INTERFACE ITF_Filling EXTENDS ITF_PackML

{warning 'add method implementation '}
METHOD Abort : BOOL
END_METHOD

{warning 'add method implementation '}
METHOD Aborting_SC : BOOL
END_METHOD

{warning 'add method implementation '}
METHOD Clear : BOOL
END_METHOD

{warning 'add method implementation '}
METHOD Clearing_SC : BOOL
END_METHOD

{warning 'add method implementation '}
METHOD Completing_SC : BOOL
END_METHOD

{warning 'add method implementation '}
METHOD Execute_SC : BOOL
END_METHOD

{warning 'add method implementation '}
METHOD FB_init : BOOL
VAR_INPUT
	bInitRetains : BOOL; // if TRUE, the retain variables are initialized (warm start / cold start)
	bInCopyCode : BOOL;  // if TRUE, the instance afterwards gets moved into the copy code (online change)
END_VAR
END_METHOD

{warning 'add method implementation '}
METHOD Hold : BOOL
END_METHOD

{warning 'add method implementation '}
METHOD Holding_SC : BOOL
END_METHOD

{warning 'add method implementation '}
METHOD Reset : BOOL
END_METHOD

{warning 'add method implementation '}
METHOD Resetting_SC : BOOL
END_METHOD

{warning 'add method implementation '}
METHOD Start : BOOL
END_METHOD

{warning 'add method implementation '}
METHOD Starting_SC : BOOL
END_METHOD

{warning 'add property implementation'}
PROPERTY State : TwinCAT_LIB.E_State_PackML
GET
END_GET
END_PROPERTY

{warning 'add method implementation '}
METHOD Stop : BOOL
END_METHOD

{warning 'add method implementation '}
METHOD Stopping_SC : BOOL
END_METHOD

{warning 'add method implementation '}
METHOD Suspend : BOOL
END_METHOD

{warning 'add method implementation '}
METHOD Suspending_SC : BOOL
END_METHOD

{warning 'add method implementation '}
METHOD Unhold : BOOL
END_METHOD

{warning 'add method implementation '}
METHOD Unholding_SC : BOOL
END_METHOD

{warning 'add method implementation '}
METHOD Unsuspend : BOOL
END_METHOD

{warning 'add method implementation '}
METHOD Unsuspending_SC : BOOL
END_METHOD

{warning 'add method implementation '}
METHOD ZeroAllVar : BOOL
END_METHOD

END_INTERFACE

(* stored: Version 1.1.0.1, ProductVersion 3.1.4024.12
   Itf ITF_Filling: Id {7e40b0bf-3742-48dd-addd-ee44a551658b}
   Folder Methods: Id {e981911d-c1d3-44f5-8ea0-c2bd3fd16631}
   Folder Properties: Id {d561a764-7773-4a8b-9f9c-0ac876449c5b}
   Method Abort: Id {1f6b5d22-314b-4c0c-a2e7-30bfd4aa7404}
   Method Aborting_SC: Id {8c463640-8115-4d8e-9408-6fc78f5520d0}
   Method Clear: Id {8a7402f5-48f6-4e75-ba75-dc97c97d40cc}
   Method Clearing_SC: Id {df617eb0-962f-455f-9c96-fb98a9fe9116}
   Method Completing_SC: Id {9dd3a585-26b4-4efe-8747-14396bcb1686}
   Method Execute_SC: Id {03c351fa-8ab7-4fb1-bfdb-913b7fc7e092}
   Method FB_init: Id {ed06c622-049c-4c15-942b-3b75d6a15d92}
   Method Hold: Id {c21bde3d-4449-41fb-af5d-0eb6bebc6196}
   Method Holding_SC: Id {2cbef641-74be-4713-9c47-c54d7a035e31}
   Method Reset: Id {669af71a-4b39-452d-a1e3-dda0848266be}
   Method Resetting_SC: Id {758ae6d7-563c-4958-bbe8-d3000b484e9d}
   Method Start: Id {9421bbf9-6722-490a-9a62-564d02602ec5}
   Method Starting_SC: Id {a1038286-50ba-404c-8bc3-ef9042dd9ee5}
   Property State: Id {d1d03dbc-0b58-45dc-8b40-a3eaa82c3c54}
   Get Get: Id {f7bf1912-d71a-4621-a347-bbab4a4e9a84}
   Method Stop: Id {8e0f6f3c-cbd2-4d6e-b40c-f84432238690}
   Method Stopping_SC: Id {c48ce6f1-8753-4401-a96f-1b8cb428b981}
   Method Suspend: Id {100b4daa-758e-4193-b8b6-78abf90f6a2d}
   Method Suspending_SC: Id {dd5eb7b5-6235-4e18-abb3-8a1e203399e0}
   Method Unhold: Id {290d9fac-4d68-48f4-8977-0a414affa371}
   Method Unholding_SC: Id {9e1b6153-236d-4d80-b225-e1252b9c843b}
   Method Unsuspend: Id {06a22e3a-bf34-4ac2-9b20-625aa98b100e}
   Method Unsuspending_SC: Id {84711ced-713c-4d89-999e-1c60665516b8}
   Method ZeroAllVar: Id {0816172b-b301-49a4-a8e1-d0bfa5a4d7c3} *)
